// TIA Portal V19 export
TYPE "LAF_typeDevDiagRisEdge"
TITLE = Edge evaluation PN device diag / Flankenauswertung PN device diag
// This data type contains the structure for edge evaluations. / PN device diag
// stored: Access Published
   STRUCT
      risEdgeManualReadAll { ExternalAccessible := 'False'; ExternalVisible := 'False'; ExternalWritable := 'False'} : Bool;   // Steigende Flanke Manueller Leseanstoss von HMI / Rising edge read from HMI manually
      posPulseManualReadAll { ExternalAccessible := 'False'; ExternalVisible := 'False'; ExternalWritable := 'False'} : Bool;   // Pos.Impuls Manueller Leseanstoss von HMI / Pos. pulse manual read from HMI
      risEdgeResetAll { ExternalAccessible := 'False'; ExternalVisible := 'False'; ExternalWritable := 'False'} : Bool;   // Steigende Flanke Reset All von HMI / Rising edge reset all from HMI
      posPulseResetAll { ExternalAccessible := 'False'; ExternalVisible := 'False'; ExternalWritable := 'False'} : Bool;   // Pos Impuls Reset All von HMI / Pos. pulse reset all
      risEdgeQuitAlarms { ExternalAccessible := 'False'; ExternalVisible := 'False'; ExternalWritable := 'False'} : Bool;   // Steigende Flanke Alarme quittieren / Rising edge reset alarm
      posPulseQuitAlarms { ExternalAccessible := 'False'; ExternalVisible := 'False'; ExternalWritable := 'False'} : Bool;   // Pos Impuls Alarme quittieren / Pos. pulse alarm reset
   END_STRUCT;
END_TYPE
